FUNCTION_BLOCK Conveyor_Model_WithNetwork (* Composite Function Block Type *)
  (* Standard: 61499-2 *)
  (* Version 0.0, 2010-12-08, User, nxtControl GmbH, template *)
  (* Compiler header: package fb.rt.cs725;import fb.rt.hmi.*; *)
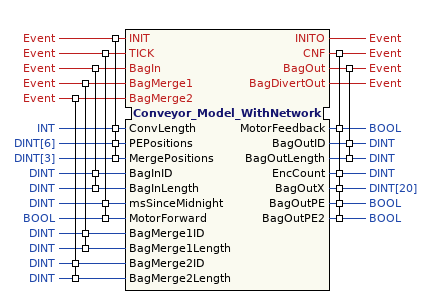
  EVENT_INPUT
    INIT WITH ConvLength, PEPositions, MergePositions; (* Initialization Request *)
    TICK WITH msSinceMidnight, MotorForward; (* Normal Execution Request *)
    BagIn WITH BagInID, BagInLength;
    BagMerge1 WITH BagMerge1ID, BagMerge1Length;
    BagMerge2 WITH BagMerge2ID, BagMerge2Length;
  END_EVENT
  EVENT_OUTPUT
    INITO; (* Initialization Confirm *)
    CNF WITH MotorFeedback, EncCount, BagOutX, BagOutPE, BagOutPE2; (* Execution Confirmation *)
    BagOut WITH BagOutID, BagOutLength;
    BagDivertOut;
  END_EVENT
  VAR_INPUT
    ConvLength : INT;
    PEPositions : ARRAY [0..5] OF DINT;
    MergePositions : ARRAY [0..2] OF DINT;
    BagInID : DINT;
    BagInLength : DINT;
    msSinceMidnight : DINT;
    MotorForward : BOOL;
    BagMerge1ID : DINT;
    BagMerge1Length : DINT;
    BagMerge2ID : DINT;
    BagMerge2Length : DINT;
  END_VAR
  VAR_OUTPUT
    MotorFeedback : BOOL;
    BagOutID : DINT;
    BagOutLength : DINT;
    EncCount : DINT;
    BagOutX : ARRAY [0..19] OF DINT;
    BagOutPE : BOOL;
    BagOutPE2 : BOOL;
  END_VAR
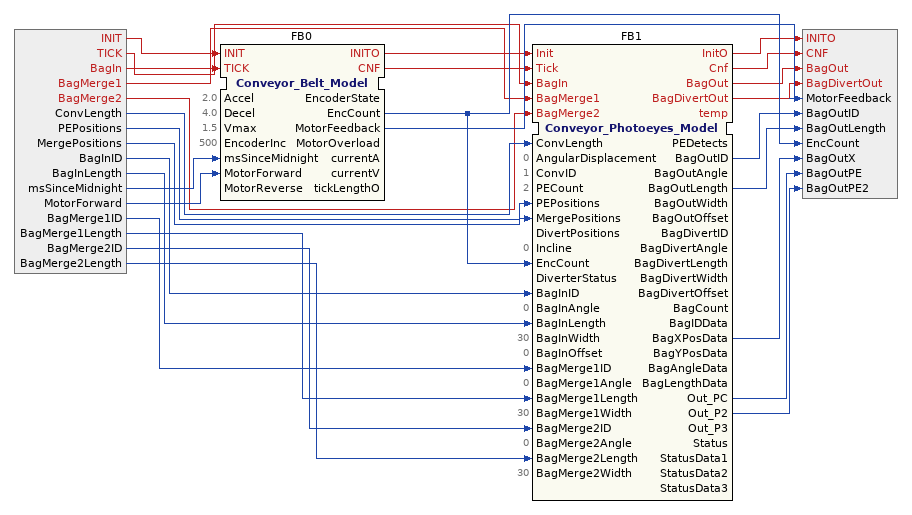
  FBS
    FB0 : Conveyor_Belt_Model(Accel := 2.0, Decel := 4.0, Vmax := 1.5, EncoderInc := 500);
    FB1 : Conveyor_Photoeyes_Model(Incline := 0, AngularDisplacement := 0, ConvID := 1, PECount := 2, BagInAngle := 0, BagInWidth := 30, BagInOffset := 0, BagMerge1Angle := 0, BagMerge1Width := 30, BagMerge2Angle := 0, BagMerge2Width := 30);
  END_FBS
  EVENT_CONNECTIONS
    INIT TO FB0.INIT;
    TICK TO FB0.TICK;
    FB0.CNF TO FB1.Tick;
    FB0.INITO TO FB1.Init;
    BagIn TO FB1.BagIn;
    FB1.BagOut TO BagOut;
    FB1.BagDivertOut TO BagDivertOut;
    BagMerge1 TO FB1.BagMerge1;
    BagMerge2 TO FB1.BagMerge2;
    FB1.InitO TO INITO;
    FB1.Cnf TO CNF;
  END_CONNECTIONS
  DATA_CONNECTIONS
    ConvLength TO FB1.ConvLength;
    PEPositions TO FB1.PEPositions;
    MergePositions TO FB1.MergePositions;
    BagInID TO FB1.BagInID;
    BagInLength TO FB1.BagInLength;
    FB1.BagOutID TO BagOutID;
    FB1.BagOutLength TO BagOutLength;
    msSinceMidnight TO FB0.msSinceMidnight;
    MotorForward TO FB0.MotorForward;
    FB0.MotorFeedback TO MotorFeedback;
    FB0.EncCount TO EncCount;
    BagMerge1ID TO FB1.BagMerge1ID;
    BagMerge1Length TO FB1.BagMerge1Length;
    BagMerge2ID TO FB1.BagMerge2ID;
    BagMerge2Length TO FB1.BagMerge2Length;
    FB1.BagXPosData TO BagOutX;
    FB1.Out_PC TO BagOutPE;
    FB0.EncCount TO FB1.EncCount;
    FB1.Out_P2 TO BagOutPE2;
  END_CONNECTIONS
END_FUNCTION_BLOCK
